PROGRAM PGR_Koffie
VAR_EXTERNAL
    bVraagKoffie  : BOOL;
    bKoffieGereed : BOOL;
END_VAR

VAR
    tKoffie : TON;
    sStatus : STRING[50];
	 iState : INT; // 0=Idle, 1=KoffieZetten, 2=Klaar
	tReis: Ton;
END_VAR

CASE iState OF

    0: // Idle
        sStatus := 'Geen koffie opdracht';
        tKoffie(IN := FALSE);
        IF bVraagKoffie THEN
            iState := 1;
        END_IF

    1: // Koffie zetten
        sStatus := 'Koffie wordt gezet';
        tKoffie(IN := TRUE, PT := T#3s);
        IF tKoffie.Q THEN
            tKoffie(IN := FALSE);
            bKoffieGereed := TRUE;
            bVraagKoffie := FALSE;
            iState := 2;
        END_IF

    2: // Klaar
        sStatus := 'Koffie is klaar';

END_CASE

END_PROGRAM

(* stored: Version 1.1.0.1, ProductVersion 3.1.4024.15
   POU PGR_Koffie: Id {7803fddf-a6de-4cbd-9adc-51c1351a8d4f}, SpecialFunc None *)
